// TIA Portal V17 export
// export: Created 2021-12-03T08:13:12.6801302Z, ExportSetting WithDefaults, DisplayName Totally Integrated Automation Portal, DisplayVersion V17, DisplayName TIA Portal Openness, DisplayVersion V17, DisplayName TIA Portal Version Control Interface, DisplayVersion V17, DisplayName STEP 7 Professional, DisplayVersion V17, DisplayName STEP 7 Safety, DisplayVersion V17, DisplayName WinCC Advanced, DisplayVersion V17
FUNCTION_BLOCK "FFB_Safety_Perimeter"   // FB300, F_FBD
VERSION : 0.1
// stored: AutoNumber false, IsIECCheckEnabled false, UDAEnableTagReadback false
   VAR_INPUT
      I_ReqAckCls : Bool;   // Запрос на закрытие периметра
      I_PrDrCls : Bool;   // Сигнал от замка о закрытии
      I_ReqCnfrm : Bool;   // Подтверждение закрытия и запрос на открытие
      I_SpRdyOpn : Bool;   // Готовность к открытию периметра
      I_AckFltRst : Bool;   // Сброс ошибки
      I_EmrStp : Bool;   // Аварийный останов
      I_KeyConv : Bool;   // Ключ конвейера
      I_SPBreak : Bool;   // Разрыв периметра нелегально
   END_VAR
   VAR_OUTPUT
      O_SPClose : Bool;   // Периметр безопасности закрыт
      O_RdySPCls_P3 : Bool;   // Готовность к закрытию периметра
      O_AckSPCls : Bool;   // Запрос на закрытие периметра
      O_OpnP : Bool;   // Происходит открытие
      O_SPBreak : Bool;
   END_VAR
   VAR DB_SPECIFIC
      S_AckSPClsP3_SR : Bool;   // Запрос на закрытие периметра P3
      S_AckSPClsP3_HIS : Bool;   // Для отслеживания переднего фронта пульт P3
   END_VAR
   VAR
      S_AckSPRst_TON { S7_SetPoint := 'True'} : TON;   // Таймер на закрытие периметра
   END_VAR
   VAR DB_SPECIFIC
      S_SP_Close_SR : Bool;   // Периметр закрыт
      S_AckSPClsP_HIS : Bool;   // Для отслеживания переднего фронта пульт P при закрытии
      S_SPBreak_SR : Bool;   // Разрыв периметра нелегально
   END_VAR
   VAR
      S_AckSPOpn_TON { S7_SetPoint := 'True'} : TON;
   END_VAR
   VAR DB_SPECIFIC
      S_AckSPOpn_SR : Bool;   // Запрос на открытие периметра
      S_AckSPOpnP_HIS : Bool;   // Для отслеживания переднего фронта пульт P при открытии
   END_VAR
   VAR_TEMP   // added for the SCL form of the ladder/FBD networks
      _w1 : Bool;
      _w2 : Bool;
   END_VAR
BEGIN

REGION Network 1: Готовность к закрытию периметра
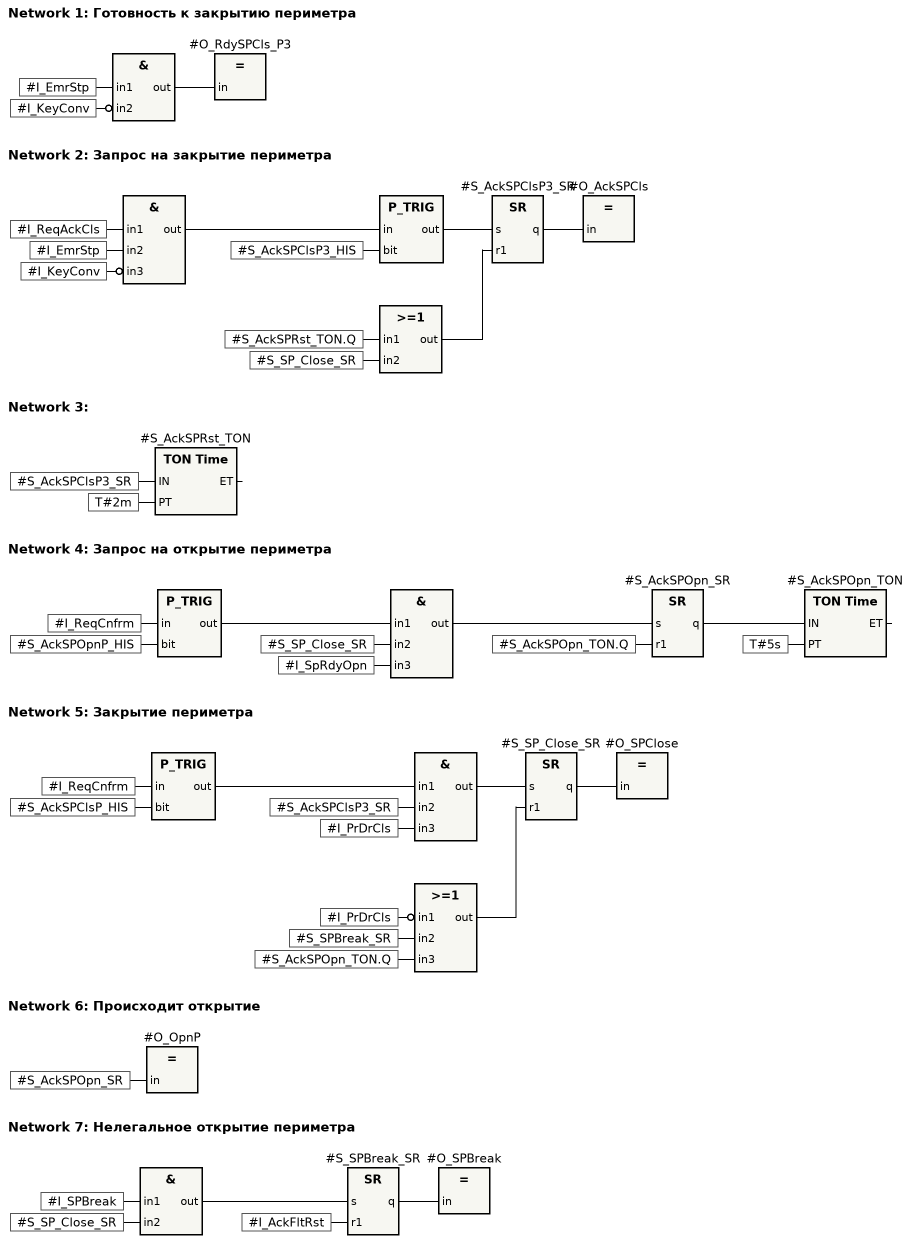
   #O_RdySPCls_P3 := #I_EmrStp AND NOT #I_KeyConv;
END_REGION

REGION Network 2: Запрос на закрытие периметра
   #_w1 := #I_ReqAckCls AND #I_EmrStp AND NOT #I_KeyConv;
   #_w2 := #_w1 AND NOT #S_AckSPClsP3_HIS;   // rising edge
   #S_AckSPClsP3_HIS := #_w1;
   IF #_w2 THEN
       #S_AckSPClsP3_SR := TRUE;   // SR flip-flop
   END_IF;
   IF #S_AckSPRst_TON.Q OR #S_SP_Close_SR THEN #S_AckSPClsP3_SR := FALSE; END_IF;
   #O_AckSPCls := #S_AckSPClsP3_SR;
END_REGION

REGION Network 3
   #S_AckSPRst_TON.TON(IN := #S_AckSPClsP3_SR, PT := T#2m);
END_REGION

REGION Network 4: Запрос на открытие периметра
   #_w1 := #I_ReqCnfrm AND NOT #S_AckSPOpnP_HIS;   // rising edge
   #S_AckSPOpnP_HIS := #I_ReqCnfrm;
   IF #_w1 AND #S_SP_Close_SR AND #I_SpRdyOpn THEN
       #S_AckSPOpn_SR := TRUE;   // SR flip-flop
   END_IF;
   IF #S_AckSPOpn_TON.Q THEN #S_AckSPOpn_SR := FALSE; END_IF;
   #S_AckSPOpn_TON.TON(IN := #S_AckSPOpn_SR, PT := T#5s);
END_REGION

REGION Network 5: Закрытие периметра
   #_w1 := #I_ReqCnfrm AND NOT #S_AckSPClsP_HIS;   // rising edge
   #S_AckSPClsP_HIS := #I_ReqCnfrm;
   IF #_w1 AND #S_AckSPClsP3_SR AND #I_PrDrCls THEN
       #S_SP_Close_SR := TRUE;   // SR flip-flop
   END_IF;
   IF NOT #I_PrDrCls OR #S_SPBreak_SR OR #S_AckSPOpn_TON.Q THEN #S_SP_Close_SR := FALSE; END_IF;
   #O_SPClose := #S_SP_Close_SR;
END_REGION

REGION Network 6: Происходит открытие
   #O_OpnP := #S_AckSPOpn_SR;
END_REGION

REGION Network 7: Нелегальное открытие периметра
   IF #I_SPBreak AND #S_SP_Close_SR THEN
       #S_SPBreak_SR := TRUE;   // SR flip-flop
   END_IF;
   IF #I_AckFltRst THEN #S_SPBreak_SR := FALSE; END_IF;
   #O_SPBreak := #S_SPBreak_SR;
END_REGION
END_FUNCTION_BLOCK
